(* LS Electric XG5000 project: 241010_1_간단한화면장치 *)
(* PLC LSPLC *)

PROGRAM NewProgram (* task: 스캔 프로그램 *)

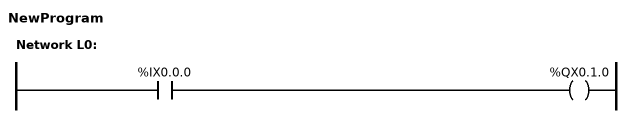
(* Rung L0 *)
%QX0.1.0 := %IX0.0.0;
END_PROGRAM